// Mitsubishi GX Works2 project: 0625(타이머_고속,저속)   PLC: Q02/Q02H

PROGRAM MAIN
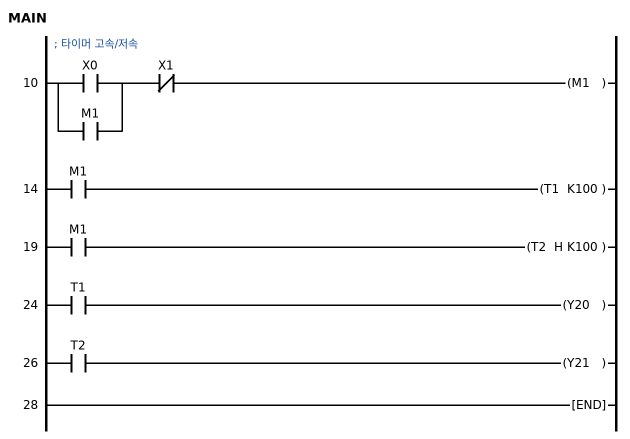
; 타이머 고속/저속
10    LD      X0
      OR      M1
      ANI     X1
      OUT     M1
14    LD      M1
      OUT     T1 K100
19    LD      M1
      OUTH    T2 K100
24    LD      T1
      OUT     Y20
26    LD      T2
      OUT     Y21
28    END
END_PROGRAM
